FUNCTION_BLOCK FB_LoadCell_Smowo_Tcp EXTENDS FB_ModbusSlaveTcp
VAR
	lrValueRaw : LREAL;
	lrValueGram : LREAL;
	lrValueKg : LREAL;
	TmpData : U_Word2Dint;
	bEnableReallyError : BOOL;
	lrRawValue : LREAL; // receive from module
	lrTareValue : LREAL; // Value at tare
END_VAR

tonConfirmReallyError(
	IN := bModbusError,
	PT := timeConfirmReallyError,
	Q => bReallyError 
);
SUPER^();

METHOD Convert : BOOL
VAR_INPUT
	iRegionNo	: 	INT;
	pReadData	:	POINTER TO word;
END_VAR
CASE iRegionNo OF
	0:
		TmpData.iWord[1] := pReadData[0];
		TmpData.iWord[0] := pReadData[1];
		lrRawValue := DINT_TO_LREAL(TmpData.idInt);
		lrValueGram :=  lrRawValue-lrTareValue;
		lrValueKg := lrValueGram * 0.001;
END_CASE
END_METHOD

PROPERTY EnableReallyError : bool
GET
EnableReallyError := bEnableReallyError;
END_GET
SET
bEnableReallyError := EnableReallyError;
END_SET
END_PROPERTY

METHOD FirstCycle // must be call once time 
VAR_INPUT
	sName : STRING;
	iUnitID : BYTE ; // modbus address of the device : 1- 255
END_VAR
THIS^.sName := sName;
THIS^.iUnitID := iUnitID;

arrAddressRead[0][0] := 0;
arrAddressRead[0][1] := 2;
arrAddressRead[0][2] := TC_ModbusBase.E_ModbusFunction.ReadHoldingRegisters;
iNumAddRegionRead := 1;
END_METHOD

PROPERTY RawValue : Lreal
GET
RawValue := lrRawValue;
END_GET
END_PROPERTY

PROPERTY TareValue : Lreal
GET
TareValue := lrTareValue;
END_GET
SET
lrTareValue := TareValue;
END_SET
END_PROPERTY

PROPERTY ValueGram : reference to lreal
GET
ValueGram REF= lrValueGram;
END_GET
END_PROPERTY

PROPERTY ValueKg : reference to lreal
GET
ValueKg ref= lrValueKg;
END_GET
END_PROPERTY

END_FUNCTION_BLOCK

(* stored: Version 1.1.0.1, ProductVersion 3.1.4024.12
   POU FB_LoadCell_Smowo_Tcp: Id {e30af404-749b-4f7c-b106-9183d8f74207}, SpecialFunc None
   Method Convert: Id {2b87e225-58d9-4340-870a-0c91076d83c2}
   Property EnableReallyError: Id {db21fd32-ad3f-46ef-9027-8fe287c987dd}
   Get Get: Id {84e1b325-f039-48a9-9898-6afd2e99d29f}
   Set Set: Id {f9faea23-9557-4776-afc8-ff3905869b35}
   Method FirstCycle: Id {f7e72015-3a1a-4225-871e-8da71edf00fc}
   Property RawValue: Id {89fdfc39-cbb7-4852-86a5-6ecdc315adfd}
   Get Get: Id {5af92946-ec89-4aeb-adb8-951a4c358a38}
   Property TareValue: Id {0b8a493a-d770-47b2-a088-28590867c0a8}
   Get Get: Id {91fc310d-da5f-43d9-8c73-180b4aef06a1}
   Set Set: Id {24d14422-496b-49a6-b957-969ed4e2b93e}
   Property ValueGram: Id {0779f1e0-95c5-4a99-9290-a85212e5d865}
   Get Get: Id {7ed4464f-d412-4f77-a082-065c61c940ca}
   Property ValueKg: Id {70ef822d-ba89-4d92-a57a-7e10348835cf}
   Get Get: Id {80fa45e1-ad71-4775-b1d9-98cc2a7b6f93} *)
